{attribute 'TcRpcEnable' := '1'}
METHOD start
  VAR_INPUT
    alphaUnits : AxesAlphaUnits;  (* The units in which alpha is given *)
    alpha : LREAL;  (* Right ascention, in the units of the alphaUnits argument *)
    deltaUnits : AxesDeltaUnits;  (* The units in which delta is given *)
    delta : LREAL;  (* Declination, in the units of the deltaUnits argument *)
    muUnits : AxesMuUnits;  (* The units in which muAlpha and muDelta are given *)
    muAlpha : LREAL;  (* Right ascention proper motion, the units of muUmits (do not multiply by cos(delta)!) *)
    muDelta : LREAL;  (* Declination proper motion, in radians/year *)
    parallax : LREAL;  (* Object parallax, in arcseconds *)
    radialVelocity : LREAL;  (* Object radial velocity, in km/s *)
    epoch : LREAL := 2000;  (* Epoch, e.g. 2000.0 *)
  END_VAR
                  THIS^.get.alphaUnits := alphaUnits;
THIS^.get.alpha := alpha;
THIS^.get.deltaUnits := deltaUnits;
THIS^.get.delta := delta;
THIS^.get.muUnits := muUnits;
THIS^.get.muAlpha := muAlpha;
THIS^.get.muDelta := muDelta;
THIS^.get.parallax := parallax;
THIS^.get.radialVelocity := radialVelocity;
THIS^.get.epoch := epoch;
THIS^.statuses.busyStatus( isBusy := TRUE );
THIS^.statuses.healthStatus( isGood := TRUE );

                
END_METHOD

{attribute 'TcRpcEnable' := '1'}
METHOD request : RequestResults
  VAR_INPUT
    alphaUnits : AxesAlphaUnits;  (* The units in which alpha is given *)
    alpha : LREAL;  (* Right ascention, in the units of the alphaUnits argument *)
    deltaUnits : AxesDeltaUnits;  (* The units in which delta is given *)
    delta : LREAL;  (* Declination, in the units of the deltaUnits argument *)
    muUnits : AxesMuUnits;  (* The units in which muAlpha and muDelta are given *)
    muAlpha : LREAL;  (* Right ascention proper motion, the units of muUmits (do not multiply by cos(delta)!) *)
    muDelta : LREAL;  (* Declination proper motion, in radians/year *)
    parallax : LREAL;  (* Object parallax, in arcseconds *)
    radialVelocity : LREAL;  (* Object radial velocity, in km/s *)
    epoch : LREAL := 2000;  (* Epoch, e.g. 2000.0 *)
  END_VAR
                  IF THIS^.statuses.enabledStatus.enabled THEN
    request := RequestResults.ACCEPTED;
    THIS^.start(
        alphaUnits := alphaUnits,
        alpha := alpha,
        deltaUnits := deltaUnits,
        delta := delta,
        muUnits := muUnits,
        muAlpha := muAlpha,
        muDelta := muDelta,
        parallax := parallax,
        radialVelocity := radialVelocity,
        epoch := epoch);
ELSE
    request := RequestResults.REJECTED;
END_IF;

                
END_METHOD
END_FUNCTION_BLOCK

FUNCTION_BLOCK AxesPointProcess EXTENDS BaseProcess
  VAR_INPUT
    state : INT;  (* State of the process *)
    {attribute 'OPC.UA.DA' := '1'}
    set : AxesPointProcessArgs;  (* Arguments to be set, before writing do_request TRUE *)
  END_VAR
  VAR_OUTPUT
    {attribute 'OPC.UA.DA' := '1'}
    {attribute 'OPC.UA.DA.Access' := '1'}
    get : AxesPointProcessArgs;  (* Arguments in use by the process, if do_request was accepted *)
  END_VAR

            IF do_request THEN
    do_request_result := request(
    alphaUnits := set.alphaUnits,
    alpha := set.alpha,
    deltaUnits := set.deltaUnits,
    delta := set.delta,
    muUnits := set.muUnits,
    muAlpha := set.muAlpha,
    muDelta := set.muDelta,
    parallax := set.parallax,
    radialVelocity := set.radialVelocity,
    epoch := set.epoch,
    tracking := set.tracking,
    rotUnits := set.rotUnits,
    rotOffset := set.rotOffset,
    rocOffset := set.rocOffset,
    ronOffset := set.ronOffset,
    doRotOffset := set.doRotOffset,
    doRocOffset := set.doRocOffset,
    doRonOffset := set.doRonOffset);
    do_request := FALSE;
END_IF;
SUPER^();

          

{attribute 'TcRpcEnable' := '1'}
METHOD start
  VAR_INPUT
    alphaUnits : AxesAlphaUnits;  (* The units in which alpha is given *)
    alpha : LREAL;  (* Right ascention, in the units of the alphaUnits argument *)
    deltaUnits : AxesDeltaUnits;  (* The units in which delta is given *)
    delta : LREAL;  (* Declination, in the units of the deltaUnits argument *)
    muUnits : AxesMuUnits;  (* The units in which muAlpha and muDelta are given *)
    muAlpha : LREAL;  (* Right ascention proper motion, the units of muUmits (do not multiply by cos(delta)!) *)
    muDelta : LREAL;  (* Declination proper motion, in radians/year *)
    parallax : LREAL;  (* Object parallax, in arcseconds *)
    radialVelocity : LREAL;  (* Object radial velocity, in km/s *)
    epoch : LREAL := 2000;  (* Epoch, e.g. 2000.0 *)
    tracking : BOOL := TRUE;  (* True to start tracking the object, false to Only do a pointing *)
    rotUnits : AxesMoveUnits;  (* Units of the 'rot', 'roc' and 'ron' arguments (RADIANS, DEGREES, ARCSECONDS, ...) *)
    rotOffset : LREAL;  (* Offset to move the currently active rotator (incompatible with 'roc' and 'ron' args) *)
    rocOffset : LREAL;  (* Offset to move the cassegrain rotation axis (incompatible with 'rot' arg) *)
    ronOffset : LREAL;  (* Offset to move the nasmyth rotation axis (incompatible with 'rot' arg) *)
    doRotOffset : BOOL;  (* True to move the currently active rotator, false to leave it untouched *)
    doRocOffset : BOOL;  (* True to move the cassegrain rotation axis, false to leave it untouched *)
    doRonOffset : BOOL;  (* True to move the nasmyth rotation axis, false to leave it untouched *)
  END_VAR
                  THIS^.get.alphaUnits := alphaUnits;
THIS^.get.alpha := alpha;
THIS^.get.deltaUnits := deltaUnits;
THIS^.get.delta := delta;
THIS^.get.muUnits := muUnits;
THIS^.get.muAlpha := muAlpha;
THIS^.get.muDelta := muDelta;
THIS^.get.parallax := parallax;
THIS^.get.radialVelocity := radialVelocity;
THIS^.get.epoch := epoch;
THIS^.get.tracking := tracking;
THIS^.get.rotUnits := rotUnits;
THIS^.get.rotOffset := rotOffset;
THIS^.get.rocOffset := rocOffset;
THIS^.get.ronOffset := ronOffset;
THIS^.get.doRotOffset := doRotOffset;
THIS^.get.doRocOffset := doRocOffset;
THIS^.get.doRonOffset := doRonOffset;
THIS^.statuses.busyStatus( isBusy := TRUE );
THIS^.statuses.healthStatus( isGood := TRUE );

                
END_METHOD

{attribute 'TcRpcEnable' := '1'}
METHOD request : RequestResults
  VAR_INPUT
    alphaUnits : AxesAlphaUnits;  (* The units in which alpha is given *)
    alpha : LREAL;  (* Right ascention, in the units of the alphaUnits argument *)
    deltaUnits : AxesDeltaUnits;  (* The units in which delta is given *)
    delta : LREAL;  (* Declination, in the units of the deltaUnits argument *)
    muUnits : AxesMuUnits;  (* The units in which muAlpha and muDelta are given *)
    muAlpha : LREAL;  (* Right ascention proper motion, the units of muUmits (do not multiply by cos(delta)!) *)
    muDelta : LREAL;  (* Declination proper motion, in radians/year *)
    parallax : LREAL;  (* Object parallax, in arcseconds *)
    radialVelocity : LREAL;  (* Object radial velocity, in km/s *)
    epoch : LREAL := 2000;  (* Epoch, e.g. 2000.0 *)
    tracking : BOOL := TRUE;  (* True to start tracking the object, false to Only do a pointing *)
    rotUnits : AxesMoveUnits;  (* Units of the 'rot', 'roc' and 'ron' arguments (RADIANS, DEGREES, ARCSECONDS, ...) *)
    rotOffset : LREAL;  (* Offset to move the currently active rotator (incompatible with 'roc' and 'ron' args) *)
    rocOffset : LREAL;  (* Offset to move the cassegrain rotation axis (incompatible with 'rot' arg) *)
    ronOffset : LREAL;  (* Offset to move the nasmyth rotation axis (incompatible with 'rot' arg) *)
    doRotOffset : BOOL;  (* True to move the currently active rotator, false to leave it untouched *)
    doRocOffset : BOOL;  (* True to move the cassegrain rotation axis, false to leave it untouched *)
    doRonOffset : BOOL;  (* True to move the nasmyth rotation axis, false to leave it untouched *)
  END_VAR
                  IF THIS^.statuses.enabledStatus.enabled THEN
    request := RequestResults.ACCEPTED;
    THIS^.start(
        alphaUnits := alphaUnits,
        alpha := alpha,
        deltaUnits := deltaUnits,
        delta := delta,
        muUnits := muUnits,
        muAlpha := muAlpha,
        muDelta := muDelta,
        parallax := parallax,
        radialVelocity := radialVelocity,
        epoch := epoch,
        tracking := tracking,
        rotUnits := rotUnits,
        rotOffset := rotOffset,
        rocOffset := rocOffset,
        ronOffset := ronOffset,
        doRotOffset := doRotOffset,
        doRocOffset := doRocOffset,
        doRonOffset := doRonOffset);
ELSE
    request := RequestResults.REJECTED;
END_IF;

                
END_METHOD
END_FUNCTION_BLOCK

FUNCTION_BLOCK AxesPointRelativeProcess EXTENDS BaseProcess
  VAR_INPUT
    {attribute 'OPC.UA.DA' := '1'}
    set : AxesPointRelativeProcessArgs;  (* Arguments to be set, before writing do_request TRUE *)
  END_VAR
  VAR_OUTPUT
    {attribute 'OPC.UA.DA' := '1'}
    {attribute 'OPC.UA.DA.Access' := '1'}
    get : AxesPointRelativeProcessArgs;  (* Arguments in use by the process, if do_request was accepted *)
  END_VAR

            IF do_request THEN
    do_request_result := request(
    alphaUnits := set.alphaUnits,
    alpha := set.alpha,
    deltaUnits := set.deltaUnits,
    delta := set.delta);
    do_request := FALSE;
END_IF;
SUPER^();

          

{attribute 'TcRpcEnable' := '1'}
METHOD start
  VAR_INPUT
    alphaUnits : AxesAlphaUnits;  (* The units in which alpha is given *)
    alpha : LREAL;  (* Right ascention, in the units of the alphaUnits argument *)
    deltaUnits : AxesDeltaUnits;  (* The units in which delta is given *)
    delta : LREAL;  (* Declination, in the units of the deltaUnits argument *)
  END_VAR
                  THIS^.get.alphaUnits := alphaUnits;
THIS^.get.alpha := alpha;
THIS^.get.deltaUnits := deltaUnits;
THIS^.get.delta := delta;
THIS^.statuses.busyStatus( isBusy := TRUE );
THIS^.statuses.healthStatus( isGood := TRUE );

                
END_METHOD

{attribute 'TcRpcEnable' := '1'}
METHOD request : RequestResults
  VAR_INPUT
    alphaUnits : AxesAlphaUnits;  (* The units in which alpha is given *)
    alpha : LREAL;  (* Right ascention, in the units of the alphaUnits argument *)
    deltaUnits : AxesDeltaUnits;  (* The units in which delta is given *)
    delta : LREAL;  (* Declination, in the units of the deltaUnits argument *)
  END_VAR
                  IF THIS^.statuses.enabledStatus.enabled THEN
    request := RequestResults.ACCEPTED;
    THIS^.start(
        alphaUnits := alphaUnits,
        alpha := alpha,
        deltaUnits := deltaUnits,
        delta := delta);
ELSE
    request := RequestResults.REJECTED;
END_IF;

                
END_METHOD
END_FUNCTION_BLOCK

FUNCTION_BLOCK AxesMoveRelativeProcess EXTENDS BaseProcess
  VAR_INPUT
    {attribute 'OPC.UA.DA' := '1'}
    set : AxesMoveRelativeProcessArgs;  (* Arguments to be set, before writing do_request TRUE *)
  END_VAR
  VAR_OUTPUT
    {attribute 'OPC.UA.DA' := '1'}
    {attribute 'OPC.UA.DA.Access' := '1'}
    get : AxesMoveRelativeProcessArgs;  (* Arguments in use by the process, if do_request was accepted *)
  END_VAR

            IF do_request THEN
    do_request_result := request(
    units := set.units,
    value := set.value);
    do_request := FALSE;
END_IF;
SUPER^();

          

{attribute 'TcRpcEnable' := '1'}
METHOD start
  VAR_INPUT
    units : AxesMoveUnits;  (* Units of the 'value' argument (RADIANS, DEGREES, ARCSECONDS, ...) *)
    value : LREAL;  (* Move the axis with this value (which units depends on the 'units' argument) *)
  END_VAR
                  THIS^.get.units := units;
THIS^.get.value := value;
THIS^.statuses.busyStatus( isBusy := TRUE );
THIS^.statuses.healthStatus( isGood := TRUE );

                
END_METHOD

{attribute 'TcRpcEnable' := '1'}
METHOD request : RequestResults
  VAR_INPUT
    units : AxesMoveUnits;  (* Units of the 'value' argument (RADIANS, DEGREES, ARCSECONDS, ...) *)
    value : LREAL;  (* Move the axis with this value (which units depends on the 'units' argument) *)
  END_VAR
                  IF THIS^.statuses.enabledStatus.enabled THEN
    request := RequestResults.ACCEPTED;
    THIS^.start(
        units := units,
        value := value);
ELSE
    request := RequestResults.REJECTED;
END_IF;

                
END_METHOD
END_FUNCTION_BLOCK

FUNCTION_BLOCK AxesMoveAbsoluteProcess EXTENDS BaseProcess
  VAR_INPUT
    {attribute 'OPC.UA.DA' := '1'}
    set : AxesMoveAbsoluteProcessArgs;  (* Arguments to be set, before writing do_request TRUE *)
  END_VAR
  VAR_OUTPUT
    {attribute 'OPC.UA.DA' := '1'}
    {attribute 'OPC.UA.DA.Access' := '1'}
    get : AxesMoveAbsoluteProcessArgs;  (* Arguments in use by the process, if do_request was accepted *)
  END_VAR

            IF do_request THEN
    do_request_result := request(
    units := set.units,
    value := set.value,
    offset := set.offset);
    do_request := FALSE;
END_IF;
SUPER^();

          

{attribute 'TcRpcEnable' := '1'}
METHOD start
  VAR_INPUT
    units : AxesMoveUnits;  (* Units of the 'value' argument (RADIANS, DEGREES, ARCSECONDS, ...) *)
    value : LREAL;  (* Move the axis to this value (which units depends on the 'units' argument) + the optional offset *)
    offset : LREAL;  (* Optional extra offset (which will not be added to the 'startPos' *)
  END_VAR
                  THIS^.get.units := units;
THIS^.get.value := value;
THIS^.get.offset := offset;
THIS^.statuses.busyStatus( isBusy := TRUE );
THIS^.statuses.healthStatus( isGood := TRUE );

                
END_METHOD

{attribute 'TcRpcEnable' := '1'}
METHOD request : RequestResults
  VAR_INPUT
    units : AxesMoveUnits;  (* Units of the 'value' argument (RADIANS, DEGREES, ARCSECONDS, ...) *)
    value : LREAL;  (* Move the axis to this value (which units depends on the 'units' argument) + the optional offset *)
    offset : LREAL;  (* Optional extra offset (which will not be added to the 'startPos' *)
  END_VAR
                  IF THIS^.statuses.enabledStatus.enabled THEN
    request := RequestResults.ACCEPTED;
    THIS^.start(
        units := units,
        value := value,
        offset := offset);
ELSE
    request := RequestResults.REJECTED;
END_IF;

                
END_METHOD
END_FUNCTION_BLOCK

FUNCTION_BLOCK AxesMoveKnownPositionProcess EXTENDS BaseProcess
  VAR_INPUT
    {attribute 'OPC.UA.DA' := '1'}
    set : AxesMoveKnownPositionProcessArgs;  (* Arguments to be set, before writing do_request TRUE *)
  END_VAR
  VAR_OUTPUT
    {attribute 'OPC.UA.DA' := '1'}
    {attribute 'OPC.UA.DA.Access' := '1'}
    get : AxesMoveKnownPositionProcessArgs;  (* Arguments in use by the process, if do_request was accepted *)
  END_VAR

            IF do_request THEN
    do_request_result := request( name := set.name );
    do_request := FALSE;
END_IF;
SUPER^();

          

{attribute 'TcRpcEnable' := '1'}
METHOD start
  VAR_INPUT
    name : STRING;  (* Name of the position to move to *)
  END_VAR
                  THIS^.get.name := name;
THIS^.statuses.busyStatus( isBusy := TRUE );
THIS^.statuses.healthStatus( isGood := TRUE );

                
END_METHOD

{attribute 'TcRpcEnable' := '1'}
METHOD request : RequestResults
  VAR_INPUT
    name : STRING;  (* Name of the position to move to *)
  END_VAR
                  IF THIS^.statuses.enabledStatus.enabled THEN
    request := RequestResults.ACCEPTED;
    THIS^.start( name := name );
ELSE
    request := RequestResults.REJECTED;
END_IF;

                
END_METHOD
END_FUNCTION_BLOCK

FUNCTION_BLOCK AxesMoveVelocityProcess EXTENDS BaseProcess
  VAR_INPUT
    {attribute 'OPC.UA.DA' := '1'}
    set : AxesMoveVelocityProcessArgs;  (* Arguments to be set, before writing do_request TRUE *)
  END_VAR
  VAR_OUTPUT
    {attribute 'OPC.UA.DA' := '1'}
    {attribute 'OPC.UA.DA.Access' := '1'}
    get : AxesMoveVelocityProcessArgs;  (* Arguments in use by the process, if do_request was accepted *)
  END_VAR

            IF do_request THEN
    do_request_result := request(
    units := set.units,
    value := set.value);
    do_request := FALSE;
END_IF;
SUPER^();

          

{attribute 'TcRpcEnable' := '1'}
METHOD start
  VAR_INPUT
    units : AxesMoveVelocityUnits;  (* Units of the 'value' argument (RADIANS_PER_SECOND, DEGREES_PER_SECOND, ...) *)
    value : LREAL;  (* Move the axis with this velocity (which units depends on the 'units' argument) *)
  END_VAR
                  THIS^.get.units := units;
THIS^.get.value := value;
THIS^.statuses.busyStatus( isBusy := TRUE );
THIS^.statuses.healthStatus( isGood := TRUE );

                
END_METHOD

{attribute 'TcRpcEnable' := '1'}
METHOD request : RequestResults
  VAR_INPUT
    units : AxesMoveVelocityUnits;  (* Units of the 'value' argument (RADIANS_PER_SECOND, DEGREES_PER_SECOND, ...) *)
    value : LREAL;  (* Move the axis with this velocity (which units depends on the 'units' argument) *)
  END_VAR
                  IF THIS^.statuses.enabledStatus.enabled THEN
    request := RequestResults.ACCEPTED;
    THIS^.start(
        units := units,
        value := value);
ELSE
    request := RequestResults.REJECTED;
END_IF;

                
END_METHOD
END_FUNCTION_BLOCK

FUNCTION_BLOCK AxesMoveOutOfLimitSwitchProcess EXTENDS BaseProcess
  VAR_INPUT
    {attribute 'OPC.UA.DA' := '1'}
    set : AxesMoveOutOfLimitSwitchProcessArgs;  (* Arguments to be set, before writing do_request TRUE *)
  END_VAR
  VAR_OUTPUT
    {attribute 'OPC.UA.DA' := '1'}
    {attribute 'OPC.UA.DA.Access' := '1'}
    get : AxesMoveOutOfLimitSwitchProcessArgs;  (* Arguments in use by the process, if do_request was accepted *)
  END_VAR

            IF do_request THEN
    do_request_result := request( switch := set.switch );
    do_request := FALSE;
END_IF;
SUPER^();

          

{attribute 'TcRpcEnable' := '1'}
METHOD start
  VAR_INPUT
    switch : LimitSwitches;  (* Positive or negative limit switch *)
  END_VAR
                  THIS^.get.switch := switch;
THIS^.statuses.busyStatus( isBusy := TRUE );
THIS^.statuses.healthStatus( isGood := TRUE );

                
END_METHOD

{attribute 'TcRpcEnable' := '1'}
METHOD request : RequestResults
  VAR_INPUT
    switch : LimitSwitches;  (* Positive or negative limit switch *)
  END_VAR
                  IF THIS^.statuses.enabledStatus.enabled THEN
    request := RequestResults.ACCEPTED;
    THIS^.start( switch := switch );
ELSE
    request := RequestResults.REJECTED;
END_IF;

                
END_METHOD
END_FUNCTION_BLOCK

FUNCTION_BLOCK AxesPowerOnProcess EXTENDS BaseProcess
  VAR_INPUT
    state : INT;  (* State of the process *)
  END_VAR

            IF do_request THEN
    do_request_result := request();
    do_request := FALSE;
END_IF;
SUPER^();

          

{attribute 'TcRpcEnable' := '1'}
METHOD start
                  THIS^.statuses.busyStatus( isBusy := TRUE );
THIS^.statuses.healthStatus( isGood := TRUE );

                
END_METHOD

{attribute 'TcRpcEnable' := '1'}
METHOD request : RequestResults
                  IF THIS^.statuses.enabledStatus.enabled THEN
    request := RequestResults.ACCEPTED;
    THIS^.start();
ELSE
    request := RequestResults.REJECTED;
END_IF;

                
END_METHOD
END_FUNCTION_BLOCK

FUNCTION_BLOCK AxesMultiPowerOnProcess EXTENDS BaseProcess
  VAR_INPUT
    state : INT;  (* State of the process *)
    {attribute 'OPC.UA.DA' := '1'}
    set : AxesMultiPowerOnProcessArgs;  (* Arguments to be set, before writing do_request TRUE *)
  END_VAR
  VAR_OUTPUT
    {attribute 'OPC.UA.DA' := '1'}
    {attribute 'OPC.UA.DA.Access' := '1'}
    get : AxesMultiPowerOnProcessArgs;  (* Arguments in use by the process, if do_request was accepted *)
  END_VAR

            IF do_request THEN
    do_request_result := request(
    azi := set.azi,
    ele := set.ele,
    roc := set.roc,
    ron := set.ron,
    fw := set.fw);
    do_request := FALSE;
END_IF;
SUPER^();

          

{attribute 'TcRpcEnable' := '1'}
METHOD start
  VAR_INPUT
    azi : BOOL;  (* TRUE to power on AZI *)
    ele : BOOL;  (* TRUE to power on ELE *)
    roc : BOOL;  (* TRUE to power on ROC *)
    ron : BOOL;  (* TRUE to power on RON *)
    fw : BOOL;  (* TRUE to power on FW *)
  END_VAR
                  THIS^.get.azi := azi;
THIS^.get.ele := ele;
THIS^.get.roc := roc;
THIS^.get.ron := ron;
THIS^.get.fw := fw;
THIS^.statuses.busyStatus( isBusy := TRUE );
THIS^.statuses.healthStatus( isGood := TRUE );

                
END_METHOD

{attribute 'TcRpcEnable' := '1'}
METHOD request : RequestResults
  VAR_INPUT
    azi : BOOL;  (* TRUE to power on AZI *)
    ele : BOOL;  (* TRUE to power on ELE *)
    roc : BOOL;  (* TRUE to power on ROC *)
    ron : BOOL;  (* TRUE to power on RON *)
    fw : BOOL;  (* TRUE to power on FW *)
  END_VAR
                  IF THIS^.statuses.enabledStatus.enabled THEN
    request := RequestResults.ACCEPTED;
    THIS^.start(
        azi := azi,
        ele := ele,
        roc := roc,
        ron := ron,
        fw := fw);
ELSE
    request := RequestResults.REJECTED;
END_IF;

                
END_METHOD
END_FUNCTION_BLOCK

FUNCTION_BLOCK AxesPowerOffProcess EXTENDS BaseProcess
  VAR_INPUT
    state : INT;  (* State of the process *)
  END_VAR

            IF do_request THEN
    do_request_result := request();
    do_request := FALSE;
END_IF;
SUPER^();

          

{attribute 'TcRpcEnable' := '1'}
METHOD start
                  THIS^.statuses.busyStatus( isBusy := TRUE );
THIS^.statuses.healthStatus( isGood := TRUE );

                
END_METHOD

{attribute 'TcRpcEnable' := '1'}
METHOD request : RequestResults
                  IF THIS^.statuses.enabledStatus.enabled THEN
    request := RequestResults.ACCEPTED;
    THIS^.start();
ELSE
    request := RequestResults.REJECTED;
END_IF;

                
END_METHOD
END_FUNCTION_BLOCK

FUNCTION_BLOCK AxesStopProcess EXTENDS BaseProcess
  VAR_INPUT
    state : INT;  (* State of the process *)
  END_VAR

            IF do_request THEN
    do_request_result := request();
    do_request := FALSE;
END_IF;
SUPER^();

          

{attribute 'TcRpcEnable' := '1'}
METHOD start
                  THIS^.statuses.busyStatus( isBusy := TRUE );
THIS^.statuses.healthStatus( isGood := TRUE );

                
END_METHOD

{attribute 'TcRpcEnable' := '1'}
METHOD request : RequestResults
                  IF THIS^.statuses.enabledStatus.enabled THEN
    request := RequestResults.ACCEPTED;
    THIS^.start();
ELSE
    request := RequestResults.REJECTED;
END_IF;

                
END_METHOD
END_FUNCTION_BLOCK

FUNCTION_BLOCK AxesSetAlphaDeltaVelocityProcess EXTENDS BaseProcess
  VAR_INPUT
    {attribute 'OPC.UA.DA' := '1'}
    set : AxesSetAlphaDeltaVelocityProcessArgs;  (* Arguments to be set, before writing do_request TRUE *)
  END_VAR
  VAR_OUTPUT
    {attribute 'OPC.UA.DA' := '1'}
    {attribute 'OPC.UA.DA.Access' := '1'}
    get : AxesSetAlphaDeltaVelocityProcessArgs;  (* Arguments in use by the process, if do_request was accepted *)
  END_VAR

            IF do_request THEN
    do_request_result := request(
    units := set.units,
    alphaVelocity := set.alphaVelocity,
    deltaVelocity := set.deltaVelocity);
    do_request := FALSE;
END_IF;
SUPER^();

          

{attribute 'TcRpcEnable' := '1'}
METHOD start
  VAR_INPUT
    units : AxesMoveVelocityUnits;  (* Units of the alphaVelocity and deltaVelocity *)
    alphaVelocity : LREAL;  (* Velocity in alpha direction *)
    deltaVelocity : LREAL;  (* Velocity in delta direction *)
  END_VAR
                  THIS^.get.units := units;
THIS^.get.alphaVelocity := alphaVelocity;
THIS^.get.deltaVelocity := deltaVelocity;
THIS^.statuses.busyStatus( isBusy := TRUE );
THIS^.statuses.healthStatus( isGood := TRUE );

                
END_METHOD

{attribute 'TcRpcEnable' := '1'}
METHOD request : RequestResults
  VAR_INPUT
    units : AxesMoveVelocityUnits;  (* Units of the alphaVelocity and deltaVelocity *)
    alphaVelocity : LREAL;  (* Velocity in alpha direction *)
    deltaVelocity : LREAL;  (* Velocity in delta direction *)
  END_VAR
                  IF THIS^.statuses.enabledStatus.enabled THEN
    request := RequestResults.ACCEPTED;
    THIS^.start(
        units := units,
        alphaVelocity := alphaVelocity,
        deltaVelocity := deltaVelocity);
ELSE
    request := RequestResults.REJECTED;
END_IF;

                
END_METHOD
END_FUNCTION_BLOCK

FUNCTION_BLOCK AxesDoHomingProcess EXTENDS BaseProcess
  VAR_INPUT
    state : INT;  (* State of the process *)
  END_VAR

            IF do_request THEN
    do_request_result := request();
    do_request := FALSE;
END_IF;
SUPER^();

          

{attribute 'TcRpcEnable' := '1'}
METHOD start
                  THIS^.statuses.busyStatus( isBusy := TRUE );
THIS^.statuses.healthStatus( isGood := TRUE );

                
END_METHOD

{attribute 'TcRpcEnable' := '1'}
METHOD request : RequestResults
                  IF THIS^.statuses.enabledStatus.enabled THEN
    request := RequestResults.ACCEPTED;
    THIS^.start();
ELSE
    request := RequestResults.REJECTED;
END_IF;

                
END_METHOD
END_FUNCTION_BLOCK

FUNCTION_BLOCK AxesMultiMoveProcess EXTENDS BaseProcess
  VAR_INPUT
    waitingForAzi : BOOL;  (* True if the process is waiting for AZI *)
    waitingForEle : BOOL;  (* True if the process is waiting for ELE *)
    waitingForRoc : BOOL;  (* True if the process is waiting for ROC *)
    waitingForRon : BOOL;  (* True if the process is waiting for RON *)
    {attribute 'OPC.UA.DA' := '1'}
    set : AxesMultiMoveProcessArgs;  (* Arguments to be set, before writing do_request TRUE *)
  END_VAR
  VAR_OUTPUT
    {attribute 'OPC.UA.DA' := '1'}
    {attribute 'OPC.UA.DA.Access' := '1'}
    get : AxesMultiMoveProcessArgs;  (* Arguments in use by the process, if do_request was accepted *)
  END_VAR

            IF do_request THEN
    do_request_result := request(
    units := set.units,
    azi := set.azi,
    ele := set.ele,
    rot := set.rot,
    roc := set.roc,
    ron := set.ron,
    doAzi := set.doAzi,
    doEle := set.doEle,
    doRot := set.doRot,
    doRoc := set.doRoc,
    doRon := set.doRon,
    preferMostTravel := set.preferMostTravel);
    do_request := FALSE;
END_IF;
SUPER^();

          

{attribute 'TcRpcEnable' := '1'}
METHOD start
  VAR_INPUT
    units : AxesMoveUnits;  (* Units of the 'azi', 'ele', 'roc' and 'ron' arguments (RADIANS, DEGREES, ARCSECONDS, ...) *)
    azi : LREAL;  (* Angle to move the azimuth axis *)
    ele : LREAL;  (* Angle to move the elevation axis *)
    rot : LREAL;  (* Angle to move the currently active rotator (incompatible with 'roc' and 'ron' args) *)
    roc : LREAL;  (* Angle to move the cassegrain rotation axis (incompatible with 'rot' arg) *)
    ron : LREAL;  (* Angle to move the nasmyth rotation axis (incompatible with 'rot' arg) *)
    doAzi : BOOL;  (* True to move the azimuth axis, false to leave it untouched *)
    doEle : BOOL;  (* True to move the elevation axis, false to leave it untouched *)
    doRot : BOOL;  (* True to move the currently active rotator, false to leave it untouched *)
    doRoc : BOOL;  (* True to move the cassegrain rotation axis, false to leave it untouched *)
    doRon : BOOL;  (* True to move the nasmyth rotation axis, false to leave it untouched *)
    preferMostTravel : BOOL := FALSE;  (* Only in case of relative movement during tracking: If possible, go to the position where there is most travel (if the telescope is tracking). If false, it will go there the quickest way possible. *)
  END_VAR
                  THIS^.get.units := units;
THIS^.get.azi := azi;
THIS^.get.ele := ele;
THIS^.get.rot := rot;
THIS^.get.roc := roc;
THIS^.get.ron := ron;
THIS^.get.doAzi := doAzi;
THIS^.get.doEle := doEle;
THIS^.get.doRot := doRot;
THIS^.get.doRoc := doRoc;
THIS^.get.doRon := doRon;
THIS^.get.preferMostTravel := preferMostTravel;
THIS^.statuses.busyStatus( isBusy := TRUE );
THIS^.statuses.healthStatus( isGood := TRUE );

                
END_METHOD

{attribute 'TcRpcEnable' := '1'}
METHOD request : RequestResults
  VAR_INPUT
    units : AxesMoveUnits;  (* Units of the 'azi', 'ele', 'roc' and 'ron' arguments (RADIANS, DEGREES, ARCSECONDS, ...) *)
    azi : LREAL;  (* Angle to move the azimuth axis *)
    ele : LREAL;  (* Angle to move the elevation axis *)
    rot : LREAL;  (* Angle to move the currently active rotator (incompatible with 'roc' and 'ron' args) *)
    roc : LREAL;  (* Angle to move the cassegrain rotation axis (incompatible with 'rot' arg) *)
    ron : LREAL;  (* Angle to move the nasmyth rotation axis (incompatible with 'rot' arg) *)
    doAzi : BOOL;  (* True to move the azimuth axis, false to leave it untouched *)
    doEle : BOOL;  (* True to move the elevation axis, false to leave it untouched *)
    doRot : BOOL;  (* True to move the currently active rotator, false to leave it untouched *)
    doRoc : BOOL;  (* True to move the cassegrain rotation axis, false to leave it untouched *)
    doRon : BOOL;  (* True to move the nasmyth rotation axis, false to leave it untouched *)
    preferMostTravel : BOOL := FALSE;  (* Only in case of relative movement during tracking: If possible, go to the position where there is most travel (if the telescope is tracking). If false, it will go there the quickest way possible. *)
  END_VAR
                  IF THIS^.statuses.enabledStatus.enabled THEN
    request := RequestResults.ACCEPTED;
    THIS^.start(
        units := units,
        azi := azi,
        ele := ele,
        rot := rot,
        roc := roc,
        ron := ron,
        doAzi := doAzi,
        doEle := doEle,
        doRot := doRot,
        doRoc := doRoc,
        doRon := doRon,
        preferMostTravel := preferMostTravel);
ELSE
    request := RequestResults.REJECTED;
END_IF;

                
END_METHOD
END_FUNCTION_BLOCK

FUNCTION_BLOCK AxesEnablePointingModelProcess EXTENDS BaseProcess
  VAR_INPUT
    {attribute 'OPC.UA.DA' := '1'}
    set : AxesEnablePointingModelProcessArgs;  (* Arguments to be set, before writing do_request TRUE *)
  END_VAR
  VAR_OUTPUT
    {attribute 'OPC.UA.DA' := '1'}
    {attribute 'OPC.UA.DA.Access' := '1'}
    get : AxesEnablePointingModelProcessArgs;  (* Arguments in use by the process, if do_request was accepted *)
  END_VAR

            IF do_request THEN
    do_request_result := request( name := set.name );
    do_request := FALSE;
END_IF;
SUPER^();

          

{attribute 'TcRpcEnable' := '1'}
METHOD start
  VAR_INPUT
    name : STRING;  (* Name of the pointing model *)
  END_VAR
                  THIS^.get.name := name;
THIS^.statuses.busyStatus( isBusy := TRUE );
THIS^.statuses.healthStatus( isGood := TRUE );

                
END_METHOD

{attribute 'TcRpcEnable' := '1'}
METHOD request : RequestResults
  VAR_INPUT
    name : STRING;  (* Name of the pointing model *)
  END_VAR
                  IF THIS^.statuses.enabledStatus.enabled THEN
    request := RequestResults.ACCEPTED;
    THIS^.start( name := name );
ELSE
    request := RequestResults.REJECTED;
END_IF;

                
END_METHOD
END_FUNCTION_BLOCK

FUNCTION_BLOCK AxesUnlockBrakeProcess EXTENDS BaseProcess
  VAR_INPUT
    {attribute 'OPC.UA.DA' := '1'}
    set : AxesUnlockBrakeProcessArgs;  (* Arguments to be set, before writing do_request TRUE *)
  END_VAR
  VAR_OUTPUT
    {attribute 'OPC.UA.DA' := '1'}
    {attribute 'OPC.UA.DA.Access' := '1'}
    get : AxesUnlockBrakeProcessArgs;  (* Arguments in use by the process, if do_request was accepted *)
  END_VAR

            IF do_request THEN
    do_request_result := request( seconds := set.seconds );
    do_request := FALSE;
END_IF;
SUPER^();

          

{attribute 'TcRpcEnable' := '1'}
METHOD start
  VAR_INPUT
    seconds : LREAL := 10.0;  (* Unlock the brake for this number of seconds (0 means forever) *)
  END_VAR
                  THIS^.get.seconds := seconds;
THIS^.statuses.busyStatus( isBusy := TRUE );
THIS^.statuses.healthStatus( isGood := TRUE );

                
END_METHOD

{attribute 'TcRpcEnable' := '1'}
METHOD request : RequestResults
  VAR_INPUT
    seconds : LREAL := 10.0;  (* Unlock the brake for this number of seconds (0 means forever) *)
  END_VAR
                  IF THIS^.statuses.enabledStatus.enabled THEN
    request := RequestResults.ACCEPTED;
    THIS^.start( seconds := seconds );
ELSE
    request := RequestResults.REJECTED;
END_IF;

                
END_METHOD
END_FUNCTION_BLOCK

FUNCTION_BLOCK AxesSetPositionProcess EXTENDS BaseProcess
  VAR_INPUT
    {attribute 'OPC.UA.DA' := '1'}
    set : AxesSetPositionProcessArgs;  (* Arguments to be set, before writing do_request TRUE *)
  END_VAR
  VAR_OUTPUT
    {attribute 'OPC.UA.DA' := '1'}
    {attribute 'OPC.UA.DA.Access' := '1'}
    get : AxesSetPositionProcessArgs;  (* Arguments in use by the process, if do_request was accepted *)
  END_VAR

            IF do_request THEN
    do_request_result := request( value := set.value );
    do_request := FALSE;
END_IF;
SUPER^();

          

{attribute 'TcRpcEnable' := '1'}
METHOD start
  VAR_INPUT
    value : LREAL;  (* New position to be taken over by the axis *)
  END_VAR
                  THIS^.get.value := value;
THIS^.statuses.busyStatus( isBusy := TRUE );
THIS^.statuses.healthStatus( isGood := TRUE );

                
END_METHOD

{attribute 'TcRpcEnable' := '1'}
METHOD request : RequestResults
  VAR_INPUT
    value : LREAL;  (* New position to be taken over by the axis *)
  END_VAR
                  IF THIS^.statuses.enabledStatus.enabled THEN
    request := RequestResults.ACCEPTED;
    THIS^.start( value := value );
ELSE
    request := RequestResults.REJECTED;
END_IF;

                
END_METHOD
END_FUNCTION_BLOCK
